Staubli VAL3: decIoWriteRequest.pgx

public program decIoWriteRequest(bool& x_bFlag (dimensions=1))
  local num l_nIndex
  local num l_nRetVal
begin
  // Copyright (c) 2016, Ocado Technology - Robotics Research Team
  //
  // Licensed under the Apache License, Version 2.0 (the "License");
  // you may not use this file except in compliance with the License.
  // You may obtain a copy of the License at
  //
  //     http://www.apache.org/licenses/LICENSE-2.0
  //
  // Unless required by applicable law or agreed to in writing, software
  // distributed under the License is distributed on an "AS IS" BASIS,
  // WITHOUT WARRANTIES OR CONDITIONS OF ANY KIND, either express or implied.
  // See the License for the specific language governing permissions and
  // limitations under the License.



  // decode message ID 65202 body (data)
  // assuming contains only one item!

  // assume failure to decode
  //rosIoWriteRequestAck.header.nReplyCode=2



  logMsg("decodeStart")




  // count
  l_nRetVal=fromBinary(rosIoWriteRequestMsg.body.nData,4,"-4l",rosIoWriteRequestMsg.ioWriteRequest.nCount)
  if (l_nRetVal!=1)
    x_bFlag=false
    return
  endIf

  logMsg("decode1")
  // type

    l_nRetVal=fromBinary(rosIoWriteRequestMsg.body.nData[4],4,"-4l",rosIoWriteRequestMsg.ioWriteRequest.nType)
    if (l_nRetVal!=1)
      x_bFlag=false
      return
    endIf

  logMsg("decode2")

  // index
  l_nRetVal=fromBinary(rosIoWriteRequestMsg.body.nData[8],4,"-4l",rosIoWriteRequestMsg.ioWriteRequest.nIndex)
  if (l_nRetVal!=1)
    x_bFlag=false
    return
  endIf

  logMsg("decode3")

  // value
  l_nRetVal=fromBinary(rosIoWriteRequestMsg.body.nData[12],4,"-4l",rosIoWriteRequestMsg.ioWriteRequest.nValue)
  if (l_nRetVal!=1)
    x_bFlag=false
    return
  endIf

  logMsg("decode success")

  // decoding successful
//  rosIoWriteReqAck.header.nReplyCode=1
//  rosIoWriteReqAck.jointTrajPt.nSeq=rosIoWriteRequestMsg.ioWriteRequest.nSeq
  x_bFlag=true
end
